// TIA Portal project "Unity-PLC" (V16)

(* hardware
DEVICE "S71500/ET200MP station_1"  S7-1500 station
   slot 0: "导轨_0"  Rack  6ES7 590-1***0-0AA0
   slot 1: "PLC_1"  CPU 1511-1 PN  6ES7 511-1AK00-0AB0  V1.8
      slot 3: "CPU 显示_1"  6ES7591-1AA00-0AA0
      slot 32768: "PROFINET 接口_1"  X1
         slot 32769: "端口_1"  X1 P1
         slot 32770: "端口_2"  X1 P2
*)

// ===== PLC "PLC_1"  CPU 1511-1 PN =====

VAR_GLOBAL   // PLC tag table "变量表_1"
   "正向启动" AT %I0.0 : Bool;
   "停止" AT %I0.1 : Bool;
   "电机正转" AT %Q0.0 : Bool;
   "电机反转" AT %Q0.1 : Bool;
   "反向启动" AT %Q0.2 : Bool;
   "上升启动" AT %I0.2 : Bool;
   "停止(1)" AT %I0.3 : Bool;
   "上升" AT %Q0.3 : Bool;
   "下降" AT %Q0.4 : Bool;
   "下降启动" AT %Q0.5 : Bool;
   "夹紧启动" AT %I0.4 : Bool;
   "停止(2)" AT %I0.5 : Bool;
   "夹紧" AT %Q0.6 : Bool;
   "放松" AT %Q0.7 : Bool;
   "放松启动" AT %Q1.0 : Bool;
   "伸出启动" AT %I0.6 : Bool;
   "停止(3)" AT %I0.7 : Bool;
   "伸出" AT %Q1.1 : Bool;
   "收回" AT %Q1.2 : Bool;
   "收回启动" AT %Q1.3 : Bool;
   "正转启动" AT %I1.0 : Bool;
   "停止(4)" AT %I1.1 : Bool;
   "正转" AT %Q1.4 : Bool;
   "反转" AT %Q1.5 : Bool;
   "反转启动" AT %Q1.6 : Bool;
   "开始" AT %I1.2 : Bool;
   "接通延时" AT %I2.0 : Bool;
   "停止(5)" AT %I2.1 : Bool;
   "停止按钮" AT %M2.2 : Bool;
   "停止按钮(1)" AT %M2.3 : Bool;
   "停止(6)" AT %I2.2 : Bool;
END_VAR

DATA_BLOCK "块_1_DB_1"   // DB1
{ S7_Optimized_Access := 'TRUE' }
VERSION : 0.1
// stored: InstanceOfName 块_1
"块_1"
BEGIN
END_DATA_BLOCK

DATA_BLOCK "块_1_DB_2"   // DB2
{ S7_Optimized_Access := 'TRUE' }
VERSION : 0.1
// stored: InstanceOfName 块_1
"块_1"
BEGIN
END_DATA_BLOCK

DATA_BLOCK "块_1_DB"   // DB3
{ S7_Optimized_Access := 'TRUE' }
VERSION : 0.1
// stored: InstanceOfName 块_1
"块_1"
BEGIN
END_DATA_BLOCK

DATA_BLOCK "块_2_DB"   // DB4
{ S7_Optimized_Access := 'TRUE' }
VERSION : 0.1
// stored: InstanceOfName 块_2
"块_2"
BEGIN
END_DATA_BLOCK

DATA_BLOCK "块_2_DB_1"   // DB5
{ S7_Optimized_Access := 'TRUE' }
VERSION : 0.1
// stored: InstanceOfName 块_2
"块_2"
BEGIN
END_DATA_BLOCK

DATA_BLOCK "块_1_DB_3"   // DB6
{ S7_Optimized_Access := 'TRUE' }
VERSION : 0.1
// stored: InstanceOfName 块_1
"块_1"
BEGIN
END_DATA_BLOCK

DATA_BLOCK "块_2_DB_2"   // DB7
{ S7_Optimized_Access := 'TRUE' }
VERSION : 0.1
// stored: InstanceOfName 块_2
"块_2"
BEGIN
END_DATA_BLOCK

DATA_BLOCK "块_2_DB_3"   // DB8
{ S7_Optimized_Access := 'TRUE' }
VERSION : 0.1
// stored: InstanceOfName 块_2
"块_2"
BEGIN
END_DATA_BLOCK

DATA_BLOCK "块_1_DB_4"   // DB9
{ S7_Optimized_Access := 'TRUE' }
VERSION : 0.1
// stored: InstanceOfName 块_1
"块_1"
BEGIN
END_DATA_BLOCK

// folder: System blocks/Program resources

DATA_BLOCK "IEC_Timer_0_DB"   // DB10
{ S7_Optimized_Access := 'TRUE' }
AUTHOR : Simatic
FAMILY : IEC
NAME : IEC_TMR
VERSION : 1.0
// stored: InstanceOfName IEC_TIMER
"IEC_TIMER"
BEGIN
END_DATA_BLOCK

DATA_BLOCK "IEC_Timer_0_DB_1"   // DB11
{ S7_Optimized_Access := 'TRUE' }
AUTHOR : Simatic
FAMILY : IEC
NAME : IEC_TMR
VERSION : 1.0
// stored: InstanceOfName IEC_TIMER
"IEC_TIMER"
BEGIN
END_DATA_BLOCK

DATA_BLOCK "IEC_Timer_0_DB_2"   // DB12
{ S7_Optimized_Access := 'TRUE' }
AUTHOR : Simatic
FAMILY : IEC
NAME : IEC_TMR
VERSION : 1.0
// stored: InstanceOfName IEC_TIMER
"IEC_TIMER"
BEGIN
END_DATA_BLOCK

DATA_BLOCK "IEC_Timer_0_DB_3"   // DB13
{ S7_Optimized_Access := 'TRUE' }
AUTHOR : Simatic
FAMILY : IEC
NAME : IEC_TMR
VERSION : 1.0
// stored: InstanceOfName IEC_TIMER
"IEC_TIMER"
BEGIN
END_DATA_BLOCK

DATA_BLOCK "IEC_Timer_0_DB_4"   // DB14
{ S7_Optimized_Access := 'TRUE' }
AUTHOR : Simatic
FAMILY : IEC
NAME : IEC_TMR
VERSION : 1.0
// stored: InstanceOfName IEC_TIMER
"IEC_TIMER"
BEGIN
END_DATA_BLOCK

DATA_BLOCK "IEC_Timer_0_DB_5"   // DB15
{ S7_Optimized_Access := 'TRUE' }
AUTHOR : Simatic
FAMILY : IEC
NAME : IEC_TMR
VERSION : 1.0
// stored: InstanceOfName IEC_TIMER
"IEC_TIMER"
BEGIN
END_DATA_BLOCK

DATA_BLOCK "IEC_Timer_0_DB_6"   // DB16
{ S7_Optimized_Access := 'TRUE' }
AUTHOR : Simatic
FAMILY : IEC
NAME : IEC_TMR
VERSION : 1.0
// stored: InstanceOfName IEC_TIMER
"IEC_TIMER"
BEGIN
END_DATA_BLOCK

// folder: (top level)

FUNCTION_BLOCK "块_1"   // FB1, GRAPH_PLUS
{ S7_Optimized_Access := 'TRUE' }
VERSION : 0.1
   VAR_INPUT
      OFF_SQ : Bool := false;   // 关闭顺控器
      INIT_SQ : Bool := false;   // 将顺序设置为初始状态
      ACK_EF : Bool := false;   // 确认所有的错误和故障
      S_PREV : Bool := false;   // 在S_NO输出参数中显示前导步
      S_NEXT : Bool := false;   // 在S_NO输出参数中显示后续步。
      SW_AUTO : Bool := false;   // 自动模式
      SW_TAP : Bool := false;   // 半自动/转换条件切换
      SW_TOP : Bool := false;   // 半自动/忽略转换条件
      SW_MAN : Bool := false;   // 手动模式
      S_SEL : Int := 0;   // 选择要在 S_NO中输出的步。
      S_ON : Bool := false;   // 激活S_NO 中显示的步。
      S_OFF : Bool := false;   // 取消激活 S_NO 中标识的步
      T_PUSH : Bool := false;   // 允许在半自动模式下跳过转换条件。
   END_VAR
   VAR_OUTPUT
      S_NO : Int := 0;   // 步编号
      S_MORE : Bool := false;   // 更多步可用，并可在S_NO中显示。
      S_ACTIVE : Bool := false;   // 在S_NO 中显示的步是激活的。
      ERR_FLT : Bool := false;   // 互锁条件或监控条件组出错
      AUTO_ON : Bool := false;   // 当前为自动模式
      TAP_ON : Bool := false;   // 已启用SW_TAP模式。
      TOP_ON : Bool := false;   // 启用半自动模式/忽略转换条件。
      MAN_ON : Bool := false;   // 已启用手动模式。
   END_VAR
   VAR
      HMI_INFO : Array[0..8] of UInt;
      IF_PAR : G7_IfParPlus_V2;
      RT_DATA : G7_RTDataPlus_V2;   // 内部数据区
      Trans1 : G7_TransitionPlus_V2;   // 转换结构
      Trans2 : G7_TransitionPlus_V2;   // 转换结构
      Trans3 : G7_TransitionPlus_V2;   // 转换结构
      Trans4 : G7_TransitionPlus_V2;   // 转换结构
      Trans5 : G7_TransitionPlus_V2;   // 转换结构
      Trans6 : G7_TransitionPlus_V2;   // 转换结构
      Trans7 : G7_TransitionPlus_V2;   // 转换结构
      Trans13 : G7_TransitionPlus_V2;   // 转换结构
      Step1 : G7_StepPlus_V2;   // 步结构
      Step2 : G7_StepPlus_V2;   // 步结构
      Step3 : G7_StepPlus_V2;   // 步结构
      Step4 : G7_StepPlus_V2;   // 步结构
      Step5 : G7_StepPlus_V2;   // 步结构
      Step6 : G7_StepPlus_V2;   // 步结构
      Step7 : G7_StepPlus_V2;   // 步结构
      Step8 : G7_StepPlus_V2;   // 步结构
      SINI : Array[0..1] of USInt;
      LSTT : Array[0..7] of USInt;
      ATAJ : Array[0..7] of USInt;
      ATAB : Array[0..7] of USInt;
      PSTT : Array[0..7] of USInt;
      NSTT : Array[0..7] of USInt;
      ASSJ : Array[0..7] of USInt;
      ASSB : Array[0..7] of USInt;
      PTTS : Array[0..7] of USInt;
      NTTS : Array[0..7] of USInt;
      SW_SQTS : Array[0..7] of USInt;
      SWITCH : Array[0..0] of USInt;
      TVX : Array[0..1] of USInt;
      TTX : Array[0..1] of USInt;
      TSX : Array[0..1] of USInt;
      S00X : Array[0..1] of USInt;
      SOFFX : Array[0..1] of USInt;
      SONX : Array[0..1] of USInt;
      SAX : Array[0..1] of USInt;
      SERRX : Array[0..8] of USInt;
      SMX : Array[0..8] of USInt;
      S0X : Array[0..8] of USInt;
      S1X : Array[0..8] of USInt;
      IL_ALARM_INST : Program_Alarm;
      SUP_ALARM_INST : Program_Alarm;
      STEP_TIME_ALARM_INST : Program_Alarm;
      IEC_TIMER_INST : IEC_TIMER;
      TRANSACTION_FLAG : Bool := false;
   END_VAR
   // SINI[0] := 2;
   // LSTT[0] := 255;
   // ATAJ[1] := 1;
   // ATAB[1] := 1;
   // PSTT[1] := 1;
   // NSTT[0] := 1;
   // ASSJ[1] := 1;
   // ASSB[1] := 1;
   // PTTS[0] := 255;
   // NTTS[1] := 1;
   // TVX[0] := 16#1;
   // TTX[0] := 16#1;
   // TSX[0] := 16#1;
   // S00X[0] := 16#1;
   // SOFFX[0] := 16#1;
   // SONX[0] := 16#1;
   // SAX[0] := 16#1;
   // SERRX[0] := 16#1;
   // SMX[0] := 16#1;
   // S0X[0] := 16#1;
   // S1X[0] := 16#1;
   // LSTT[1] := 255;
   // LSTT[2] := 255;
   // LSTT[3] := 255;
   // LSTT[4] := 255;
   // LSTT[5] := 255;
   // LSTT[6] := 255;
   // ATAJ[2] := 2;
   // ATAJ[3] := 3;
   // ATAJ[4] := 4;
   // ATAJ[5] := 5;
   // ATAJ[6] := 6;
   // ATAJ[7] := 7;
   // ATAB[2] := 2;
   // ATAB[3] := 3;
   // ATAB[4] := 4;
   // ATAB[5] := 5;
   // ATAB[6] := 6;
   // ATAB[7] := 7;
   // PSTT[2] := 2;
   // PSTT[3] := 3;
   // PSTT[4] := 4;
   // PSTT[5] := 5;
   // PSTT[6] := 6;
   // PSTT[7] := 7;
   // NSTT[1] := 2;
   // NSTT[2] := 3;
   // NSTT[3] := 4;
   // NSTT[4] := 5;
   // NSTT[5] := 6;
   // NSTT[6] := 7;
   // ASSJ[2] := 2;
   // ASSJ[3] := 3;
   // ASSJ[4] := 4;
   // ASSJ[5] := 5;
   // ASSJ[6] := 6;
   // ASSJ[7] := 7;
   // ASSB[2] := 2;
   // ASSB[3] := 3;
   // ASSB[4] := 4;
   // ASSB[5] := 5;
   // ASSB[6] := 6;
   // ASSB[7] := 7;
   // PTTS[2] := 1;
   // PTTS[3] := 2;
   // PTTS[4] := 3;
   // PTTS[5] := 4;
   // PTTS[6] := 5;
   // PTTS[7] := 6;
   // NTTS[2] := 2;
   // NTTS[3] := 3;
   // NTTS[4] := 4;
   // NTTS[5] := 5;
   // NTTS[6] := 6;
   // NTTS[7] := 7;
BEGIN
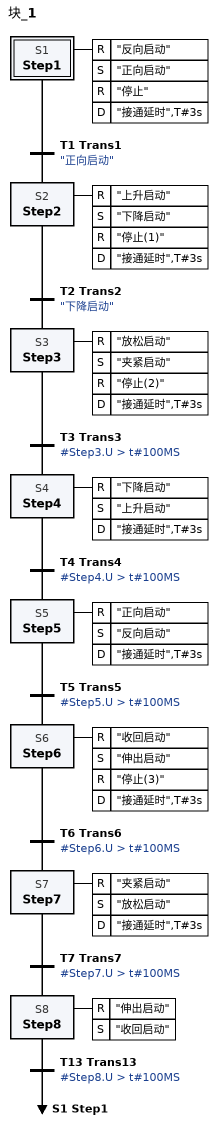
   // sequencer 1
   INITIAL_STEP Step1:   // S1, max time T#10S, warning time T#7S
              R    "反向启动"
              S    "正向启动"
              R    "停止"
              D    "接通延时",T#3s
   END_STEP
   TRANSITION Trans1 FROM Step1 TO Step2   // T1
      := "正向启动";
   END_TRANSITION
   STEP Step2:   // S2, max time T#10S, warning time T#7S
              R    "上升启动"
              S    "下降启动"
              R    "停止(1)"
              D    "接通延时",T#3s
   END_STEP
   TRANSITION Trans2 FROM Step2 TO Step3   // T2
      := "下降启动";
   END_TRANSITION
   STEP Step3:   // S3, max time T#10S, warning time T#7S
              R    "放松启动"
              S    "夹紧启动"
              R    "停止(2)"
              D    "接通延时",T#3s
   END_STEP
   TRANSITION Trans3 FROM Step3 TO Step4   // T3
      := #Step3.U > t#100MS;
   END_TRANSITION
   STEP Step4:   // S4, max time T#10S, warning time T#7S
              R    "下降启动"
              S    "上升启动"
              D    "接通延时",T#3s
   END_STEP
   TRANSITION Trans4 FROM Step4 TO Step5   // T4
      := #Step4.U > t#100MS;
   END_TRANSITION
   STEP Step5:   // S5, max time T#10S, warning time T#7S
              R    "正向启动"
              S    "反向启动"
              D    "接通延时",T#3s
   END_STEP
   TRANSITION Trans5 FROM Step5 TO Step6   // T5
      := #Step5.U > t#100MS;
   END_TRANSITION
   STEP Step6:   // S6, max time T#10S, warning time T#7S
              R    "收回启动"
              S    "伸出启动"
              R    "停止(3)"
              D    "接通延时",T#3s
   END_STEP
   TRANSITION Trans6 FROM Step6 TO Step7   // T6
      := #Step6.U > t#100MS;
   END_TRANSITION
   STEP Step7:   // S7, max time T#10S, warning time T#7S
              R    "夹紧启动"
              S    "放松启动"
              D    "接通延时",T#3s
   END_STEP
   TRANSITION Trans7 FROM Step7 TO Step8   // T7
      := #Step7.U > t#100MS;
   END_TRANSITION
   STEP Step8:   // S8, max time T#10S, warning time T#7S
              R    "伸出启动"
              S    "收回启动"
   END_STEP
   TRANSITION Trans13 FROM Step8 TO Step1   // T13, jump
      := #Step8.U > t#100MS;
   END_TRANSITION
END_FUNCTION_BLOCK

FUNCTION_BLOCK "块_2"   // FB2, GRAPH_PLUS
{ S7_Optimized_Access := 'TRUE' }
VERSION : 0.1
   VAR_INPUT
      OFF_SQ : Bool := false;   // 关闭顺控器
      INIT_SQ : Bool := false;   // 将顺序设置为初始状态
      ACK_EF : Bool := false;   // 确认所有的错误和故障
      S_PREV : Bool := false;   // 在S_NO输出参数中显示前导步
      S_NEXT : Bool := false;   // 在S_NO输出参数中显示后续步。
      SW_AUTO : Bool := false;   // 自动模式
      SW_TAP : Bool := false;   // 半自动/转换条件切换
      SW_TOP : Bool := false;   // 半自动/忽略转换条件
      SW_MAN : Bool := false;   // 手动模式
      S_SEL : Int := 0;   // 选择要在 S_NO中输出的步。
      S_ON : Bool := false;   // 激活S_NO 中显示的步。
      S_OFF : Bool := false;   // 取消激活 S_NO 中标识的步
      T_PUSH : Bool := false;   // 允许在半自动模式下跳过转换条件。
   END_VAR
   VAR_OUTPUT
      S_NO : Int := 0;   // 步编号
      S_MORE : Bool := false;   // 更多步可用，并可在S_NO中显示。
      S_ACTIVE : Bool := false;   // 在S_NO 中显示的步是激活的。
      ERR_FLT : Bool := false;   // 互锁条件或监控条件组出错
      AUTO_ON : Bool := false;   // 当前为自动模式
      TAP_ON : Bool := false;   // 已启用SW_TAP模式。
      TOP_ON : Bool := false;   // 启用半自动模式/忽略转换条件。
      MAN_ON : Bool := false;   // 已启用手动模式。
   END_VAR
   VAR
      HMI_INFO : Array[0..8] of UInt;
      IF_PAR : G7_IfParPlus_V2;
      RT_DATA : G7_RTDataPlus_V2;   // 内部数据区
      Trans1 : G7_TransitionPlus_V2;   // 转换结构
      Trans2 : G7_TransitionPlus_V2;   // 转换结构
      Trans3 : G7_TransitionPlus_V2;   // 转换结构
      Step2 : G7_StepPlus_V2;   // 步结构
      Step3 : G7_StepPlus_V2;   // 步结构
      Step4 : G7_StepPlus_V2;   // 步结构
      SINI : Array[0..1] of USInt;
      LSTT : Array[0..2] of USInt;
      ATAJ : Array[0..2] of USInt;
      ATAB : Array[0..2] of USInt;
      PSTT : Array[0..2] of USInt;
      NSTT : Array[0..2] of USInt;
      ASSJ : Array[0..2] of USInt;
      ASSB : Array[0..2] of USInt;
      PTTS : Array[0..2] of USInt;
      NTTS : Array[0..2] of USInt;
      SW_SQTS : Array[0..2] of USInt;
      SWITCH : Array[0..0] of USInt;
      TVX : Array[0..1] of USInt;
      TTX : Array[0..1] of USInt;
      TSX : Array[0..1] of USInt;
      S00X : Array[0..1] of USInt;
      SOFFX : Array[0..1] of USInt;
      SONX : Array[0..1] of USInt;
      SAX : Array[0..1] of USInt;
      SERRX : Array[0..3] of USInt;
      SMX : Array[0..3] of USInt;
      S0X : Array[0..3] of USInt;
      S1X : Array[0..3] of USInt;
      IL_ALARM_INST : Program_Alarm;
      SUP_ALARM_INST : Program_Alarm;
      STEP_TIME_ALARM_INST : Program_Alarm;
      IEC_TIMER_INST : IEC_TIMER;
      TRANSACTION_FLAG : Bool := false;
   END_VAR
   // SINI[0] := 2;
   // LSTT[0] := 255;
   // LSTT[1] := 255;
   // ATAJ[1] := 1;
   // ATAJ[2] := 2;
   // ATAB[1] := 1;
   // ATAB[2] := 2;
   // PSTT[1] := 1;
   // PSTT[2] := 2;
   // NSTT[0] := 1;
   // NSTT[1] := 2;
   // ASSJ[1] := 1;
   // ASSJ[2] := 2;
   // ASSB[1] := 1;
   // ASSB[2] := 2;
   // PTTS[0] := 255;
   // PTTS[2] := 1;
   // NTTS[1] := 1;
   // NTTS[2] := 2;
   // TVX[0] := 16#1;
   // TTX[0] := 16#1;
   // TSX[0] := 16#1;
   // S00X[0] := 16#1;
   // SOFFX[0] := 16#1;
   // SONX[0] := 16#1;
   // SAX[0] := 16#1;
   // SERRX[0] := 16#1;
   // SMX[0] := 16#1;
   // S0X[0] := 16#1;
   // S1X[0] := 16#1;
BEGIN
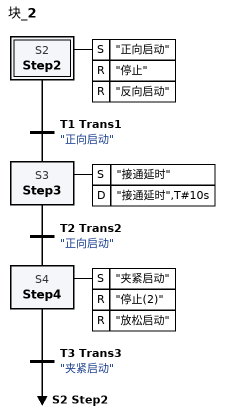
   // sequencer 1
   INITIAL_STEP Step2:   // S2, max time T#10S, warning time T#7S
              S    "正向启动"
              R    "停止"
              R    "反向启动"
   END_STEP
   TRANSITION Trans1 FROM Step2 TO Step3   // T1
      := "正向启动";
   END_TRANSITION
   STEP Step3:   // S3, max time T#10S, warning time T#7S
              S    "接通延时"
              D    "接通延时",T#10s
   END_STEP
   TRANSITION Trans2 FROM Step3 TO Step4   // T2
      := "正向启动";
   END_TRANSITION
   STEP Step4:   // S4, max time T#10S, warning time T#7S
              S    "夹紧启动"
              R    "停止(2)"
              R    "放松启动"
   END_STEP
   TRANSITION Trans3 FROM Step4 TO Step2   // T3, jump
      := "夹紧启动";
   END_TRANSITION
END_FUNCTION_BLOCK

ORGANIZATION_BLOCK "Main"   // OB1, LAD, ProgramCycle
TITLE = "Main Program Sweep (Cycle)"
{ S7_Optimized_Access := 'TRUE' }
VERSION : 0.1
   VAR_INPUT
      Initial_Call : Bool;   // Initial call of this OB
      Remanence : Bool;   // =True, if remanent data are available
   END_VAR
BEGIN
END_ORGANIZATION_BLOCK

ORGANIZATION_BLOCK "Main_1"   // OB123, LAD, ProgramCycle
TITLE = "Main Program Sweep (Cycle)"
{ S7_Optimized_Access := 'TRUE' }
VERSION : 0.1
   VAR_INPUT
      Initial_Call : Bool;   // Initial call of this OB
      Remanence : Bool;   // =True, if remanent data are available
   END_VAR
BEGIN

REGION Network 1
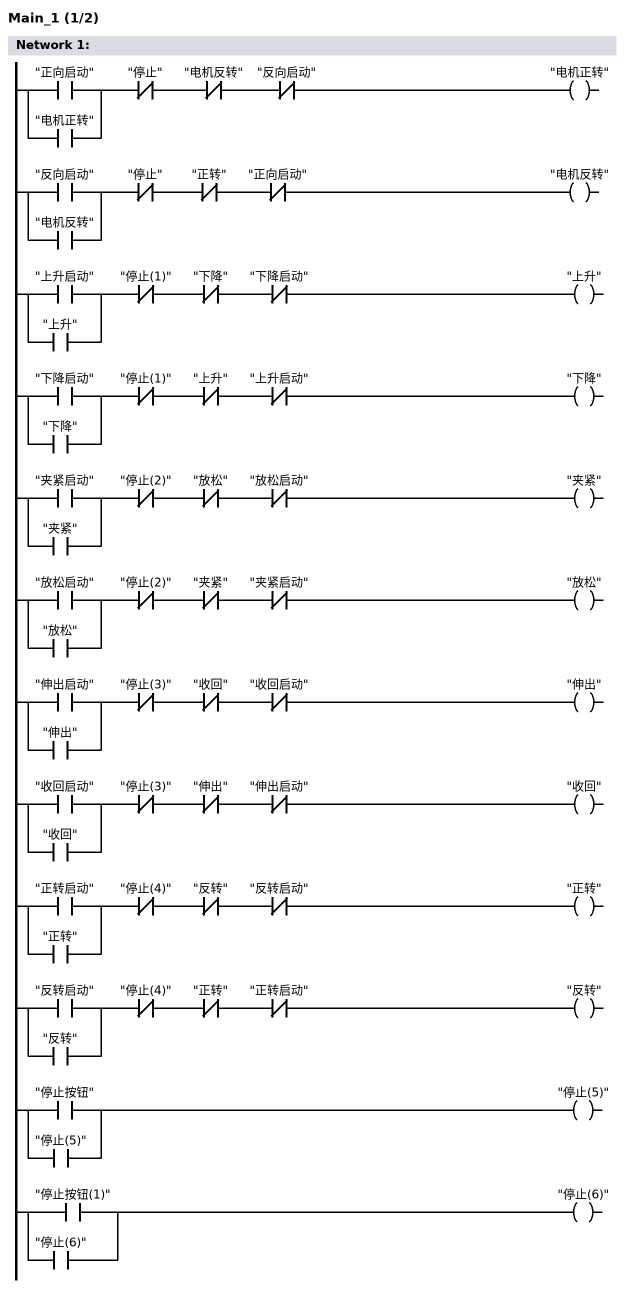
   RUNG wire#powerrail
      Contact( "正向启动" )
      wire#w1
      I_Contact( "停止" )
      I_Contact( "电机反转" )
      I_Contact( "反向启动" )
      Coil( "电机正转" )
   END_RUNG
   RUNG wire#powerrail
      Contact( "电机正转" )
   END_RUNG wire#w1
   RUNG wire#powerrail
      Contact( "反向启动" )
      wire#w2
      I_Contact( "停止" )
      I_Contact( "正转" )
      I_Contact( "正向启动" )
      Coil( "电机反转" )
   END_RUNG
   RUNG wire#powerrail
      Contact( "电机反转" )
   END_RUNG wire#w2
   RUNG wire#powerrail
      Contact( "上升启动" )
      wire#w3
      I_Contact( "停止(1)" )
      I_Contact( "下降" )
      I_Contact( "下降启动" )
      Coil( "上升" )
   END_RUNG
   RUNG wire#powerrail
      Contact( "上升" )
   END_RUNG wire#w3
   RUNG wire#powerrail
      Contact( "下降启动" )
      wire#w4
      I_Contact( "停止(1)" )
      I_Contact( "上升" )
      I_Contact( "上升启动" )
      Coil( "下降" )
   END_RUNG
   RUNG wire#powerrail
      Contact( "下降" )
   END_RUNG wire#w4
   RUNG wire#powerrail
      Contact( "夹紧启动" )
      wire#w5
      I_Contact( "停止(2)" )
      I_Contact( "放松" )
      I_Contact( "放松启动" )
      Coil( "夹紧" )
   END_RUNG
   RUNG wire#powerrail
      Contact( "夹紧" )
   END_RUNG wire#w5
   RUNG wire#powerrail
      Contact( "放松启动" )
      wire#w6
      I_Contact( "停止(2)" )
      I_Contact( "夹紧" )
      I_Contact( "夹紧启动" )
      Coil( "放松" )
   END_RUNG
   RUNG wire#powerrail
      Contact( "放松" )
   END_RUNG wire#w6
   RUNG wire#powerrail
      Contact( "伸出启动" )
      wire#w7
      I_Contact( "停止(3)" )
      I_Contact( "收回" )
      I_Contact( "收回启动" )
      Coil( "伸出" )
   END_RUNG
   RUNG wire#powerrail
      Contact( "伸出" )
   END_RUNG wire#w7
   RUNG wire#powerrail
      Contact( "收回启动" )
      wire#w8
      I_Contact( "停止(3)" )
      I_Contact( "伸出" )
      I_Contact( "伸出启动" )
      Coil( "收回" )
   END_RUNG
   RUNG wire#powerrail
      Contact( "收回" )
   END_RUNG wire#w8
   RUNG wire#powerrail
      Contact( "正转启动" )
      wire#w9
      I_Contact( "停止(4)" )
      I_Contact( "反转" )
      I_Contact( "反转启动" )
      Coil( "正转" )
   END_RUNG
   RUNG wire#powerrail
      Contact( "正转" )
   END_RUNG wire#w9
   RUNG wire#powerrail
      Contact( "反转启动" )
      wire#w10
      I_Contact( "停止(4)" )
      I_Contact( "正转" )
      I_Contact( "正转启动" )
      Coil( "反转" )
   END_RUNG
   RUNG wire#powerrail
      Contact( "反转" )
   END_RUNG wire#w10
   RUNG wire#powerrail
      Contact( "停止按钮" )
      wire#w11
      Coil( "停止(5)" )
   END_RUNG
   RUNG wire#powerrail
      Contact( "停止(5)" )
   END_RUNG wire#w11
   RUNG wire#powerrail
      Contact( "停止按钮(1)" )
      wire#w12
      Coil( "停止(6)" )
   END_RUNG
   RUNG wire#powerrail
      Contact( "停止(6)" )
   END_RUNG wire#w12
   // the same network as SCL:
   "电机正转" := ("正向启动" OR "电机正转") AND NOT "停止" AND NOT "电机反转" AND NOT "反向启动";
   "电机反转" := ("反向启动" OR "电机反转") AND NOT "停止" AND NOT "正转" AND NOT "正向启动";
   "上升" := ("上升启动" OR "上升") AND NOT "停止(1)" AND NOT "下降" AND NOT "下降启动";
   "下降" := ("下降启动" OR "下降") AND NOT "停止(1)" AND NOT "上升" AND NOT "上升启动";
   "夹紧" := ("夹紧启动" OR "夹紧") AND NOT "停止(2)" AND NOT "放松" AND NOT "放松启动";
   "放松" := ("放松启动" OR "放松") AND NOT "停止(2)" AND NOT "夹紧" AND NOT "夹紧启动";
   "伸出" := ("伸出启动" OR "伸出") AND NOT "停止(3)" AND NOT "收回" AND NOT "收回启动";
   "收回" := ("收回启动" OR "收回") AND NOT "停止(3)" AND NOT "伸出" AND NOT "伸出启动";
   "正转" := ("正转启动" OR "正转") AND NOT "停止(4)" AND NOT "反转" AND NOT "反转启动";
   "反转" := ("反转启动" OR "反转") AND NOT "停止(4)" AND NOT "正转" AND NOT "正转启动";
   "停止(5)" := "停止按钮" OR "停止(5)";
   "停止(6)" := "停止按钮(1)" OR "停止(6)";
END_REGION

REGION Network 2
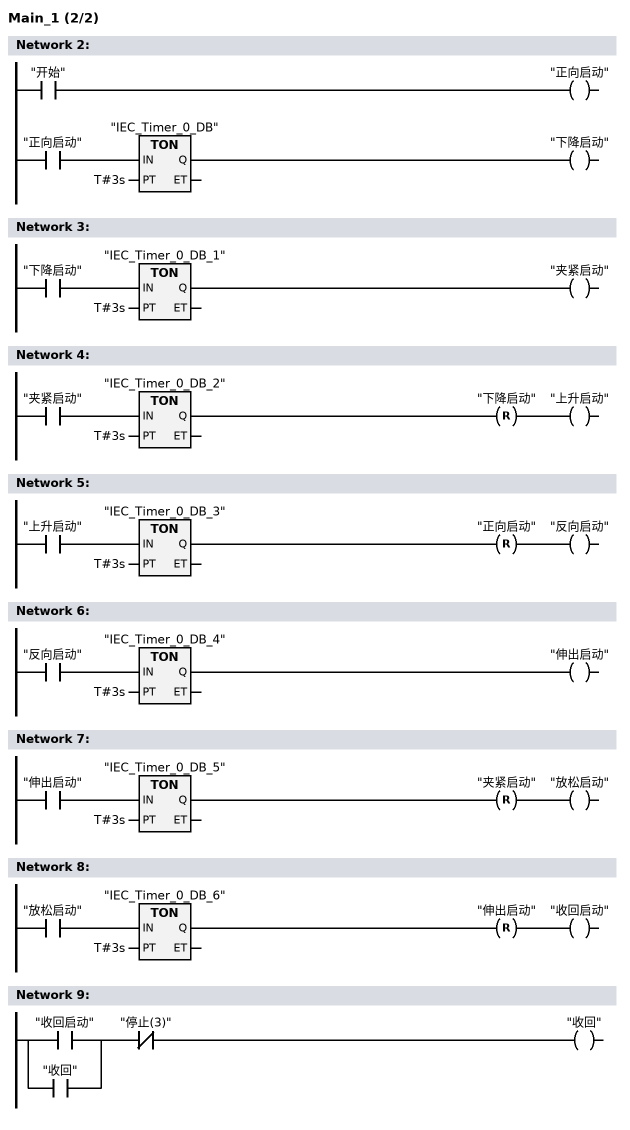
   "正向启动" := "开始";
   "IEC_Timer_0_DB".TON(IN := "正向启动", PT := T#3s);
   "下降启动" := "IEC_Timer_0_DB".Q;
END_REGION

REGION Network 3
   "IEC_Timer_0_DB_1".TON(IN := "下降启动", PT := T#3s);
   "夹紧启动" := "IEC_Timer_0_DB_1".Q;
END_REGION

REGION Network 4
   "IEC_Timer_0_DB_2".TON(IN := "夹紧启动", PT := T#3s);
   IF "IEC_Timer_0_DB_2".Q THEN "下降启动" := FALSE; END_IF;
   "上升启动" := "IEC_Timer_0_DB_2".Q;
END_REGION

REGION Network 5
   "IEC_Timer_0_DB_3".TON(IN := "上升启动", PT := T#3s);
   IF "IEC_Timer_0_DB_3".Q THEN "正向启动" := FALSE; END_IF;
   "反向启动" := "IEC_Timer_0_DB_3".Q;
END_REGION

REGION Network 6
   "IEC_Timer_0_DB_4".TON(IN := "反向启动", PT := T#3s);
   "伸出启动" := "IEC_Timer_0_DB_4".Q;
END_REGION

REGION Network 7
   "IEC_Timer_0_DB_5".TON(IN := "伸出启动", PT := T#3s);
   IF "IEC_Timer_0_DB_5".Q THEN "夹紧启动" := FALSE; END_IF;
   "放松启动" := "IEC_Timer_0_DB_5".Q;
END_REGION

REGION Network 8
   "IEC_Timer_0_DB_6".TON(IN := "放松启动", PT := T#3s);
   IF "IEC_Timer_0_DB_6".Q THEN "伸出启动" := FALSE; END_IF;
   "收回启动" := "IEC_Timer_0_DB_6".Q;
END_REGION

REGION Network 9
   RUNG wire#powerrail
      Contact( "收回启动" )
      wire#w1
      I_Contact( "停止(3)" )
      Coil( "收回" )
   END_RUNG
   RUNG wire#powerrail
      Contact( "收回" )
   END_RUNG wire#w1
   // the same network as SCL:
   "收回" := ("收回启动" OR "收回") AND NOT "停止(3)";
END_REGION
END_ORGANIZATION_BLOCK